// TIA Portal V19 export
DATA_BLOCK "A0302_Rulliera"   // DB85
// stored: InstanceOfName A0302_Rulliera_FB, InstanceOfType FB
"A0302_Rulliera_FB"
   // VAR_INPUT
   //    AreaInterface : "AreaInterface";
   //    ZSI : "udt_ZoneSafetyInterface";
   //    DSI_Feed1 : "udt_DeviceSafetyInterface";
   //    DSI_Feed2 : "udt_DeviceSafetyInterface";
   //    Drive_Ax1 : "TAx_DriveInterface";
   //    Drive_Ax2 : "TAx_DriveInterface";
   //    DataIn : Struct
   //       Ax : "SpeedMachine_DataIn";
   //       Sens : Struct
   //          Coda { ExternalAccessible := 'False'; ExternalVisible := 'False'; ExternalWritable := 'False'} : Struct
   //             FTC_Rall : Bool;
   //             FTC_Prox_Ing : Bool;
   //          END_STRUCT;
   //          Centro { ExternalAccessible := 'False'; ExternalVisible := 'False'; ExternalWritable := 'False'} : Struct
   //             FTC_Centrale : Bool;
   //          END_STRUCT;
   //       END_STRUCT;
   //    END_STRUCT;
   //    CIn { ExternalAccessible := 'False'; ExternalVisible := 'False'; ExternalWritable := 'False'} : Struct
   //       Manager : Struct
   //          Ax_1 : "SpeedMachine_CIn_Manager";
   //          Ax_2 : "SpeedMachine_CIn_Manager";
   //       END_STRUCT;
   //       SemiAut_Pb : Bool;
   //       P5 : Struct
   //          Sollevatori : "ValveMachine_COut";
   //          SpintoreLong : "ValveMachine_COut";
   //          Sens : Struct
   //             FTC_Ingombro_A0301 : Bool;
   //          END_STRUCT;
   //       END_STRUCT;
   //       Bordatrice : Struct
   //          StopBordatrice : Bool;
   //          ReadyForMove : Bool;
   //          StandbyBordatrice : Bool;
   //       END_STRUCT;
   //       Rulliera : Struct
   //          Centratori : "ValveMachine_COut";
   //          Sollevamento : "ValveMachine_COut";
   //          Coda : Struct
   //             Sens : Struct
   //                FTC_Rall : Bool;
   //                FTC_Prox_Ing : Bool;
   //             END_STRUCT;
   //          END_STRUCT;
   //          Centro : Struct
   //             Sens : Struct
   //                FTC_Centrale : Bool;
   //             END_STRUCT;
   //          END_STRUCT;
   //       END_STRUCT;
   //       CarroPareggCoda : Struct
   //          Ax : "Positioning_DOL_Machine_COut";
   //          Bloccaggio : "ValveMachine_COut";
   //          BattutaVerticale : "ValveMachine_COut";
   //          PareggiatoreLong : "ValveMachine_COut";
   //          Sens : Struct
   //             FTC_Ingombro_In : Bool;
   //             FTC_Ingombro_Out : Bool;
   //             PresenzaMat : Bool;
   //             PosPareggLong : Struct
   //                Value : LReal;
   //                CheckMeasure : Bool;
   //                Standstill : Bool;
   //             END_STRUCT;
   //          END_STRUCT;
   //       END_STRUCT;
   //       CarroPareggTesta : Struct
   //          Ax : "Positioning_DOL_Machine_COut";
   //          Bloccaggio : "ValveMachine_COut";
   //          Centraggio : "ValveMachine_COut";
   //          Sollevatore : "ValveMachine_COut";
   //          Sens : Struct
   //             FTC1_Rall : Bool;
   //             FTC2_Prox_Ls : Bool;
   //             PresenzaMat : Bool;
   //          END_STRUCT;
   //       END_STRUCT;
   //       BTrk : Struct
   //          ZoneA0302Entry_Empty : Bool;
   //          ZoneA0302Exit_Empty : Bool;
   //       END_STRUCT;
   //    END_STRUCT;
   //    Config : Struct
   //       Ax : "SpeedMachine_Config";
   //    END_STRUCT;
   //    HWID_Ax_TEL1 : Array[1..2] of HW_SUBMODULE;
   // END_VAR
   // VAR_OUTPUT
   //    MachineInterface : "MachineInterface";
   //    COut : Struct
   //       Ax_1 : "SpeedMachine_COut";
   //       Ax_2 : "SpeedMachine_COut";
   //       Ax_VelOveride : Struct
   //          Enable : Bool;
   //          Value : Real;
   //       END_STRUCT;
   //    END_STRUCT;
   // END_VAR
   // VAR_IN_OUT
   //    Par : Struct
   //       Ax : "SpeedMachine_Par";
   //       Ax_Aut : "A0301_Mach_Speed_Par";
   //    END_STRUCT;
   //    IEC_SP : Struct
   //       FTC_CodaRall : Struct
   //          TON_PT : Time;
   //          TOF_PT : Time;
   //       END_STRUCT;
   //       FTC_CodaProx_Ing : Struct
   //          TON_PT : Time;
   //          TOF_PT : Time;
   //       END_STRUCT;
   //       FTC_Centro : Struct
   //          TON_PT : Time;
   //          TOF_PT : Time;
   //       END_STRUCT;
   //    END_STRUCT;
   // END_VAR
   // VAR
   //    Alarm : Struct
   //       Rulliera : Array[1..2] of "SpeedMachine_Alr";
   //    END_STRUCT;
   //    Warning : Struct
   //       Rulliera : Array[1..2] of "SpeedMachine_Wng";
   //       OP_REST_MissingCnd : Bool;
   //       OP_WORK_MissingCnd : Bool;
   //    END_STRUCT;
   //    HMI : Struct
   //       Selection : Struct
   //          Ax : Int;
   //       END_STRUCT;
   //    END_STRUCT;
   //    Ax_1 : "SpeedMachine_FB";
   //    Ax_2 : "SpeedMachine_FB";
   //    ValueVelOvr { ExternalAccessible := 'False'; ExternalVisible := 'False'; ExternalWritable := 'False'} : Array[1..10] of Real;
   //    Sts : Struct
   //       OP_CanMoveFreely : Bool;
   //       OP_Bwd_Cnd : Bool;
   //       OP_Fwd_Cnd : Bool;
   //    END_STRUCT;
   //    Ctrl : Struct
   //       OP_Bwd_Man : Bool;
   //       OP_Fwd_Man : Bool;
   //       OP_Bwd_Aut : Bool;
   //       OP_Fwd_Aut : Bool;
   //       OP_Bwd_Run : Bool;
   //       OP_Fwd_Run : Bool;
   //    END_STRUCT;
   //    AUX : Struct
   //       OP_Bwd_PB : Bool;
   //       OP_Fwd_PB : Bool;
   //    END_STRUCT;
   //    TON_OP_REST_MissingCnd { S7_SetPoint := 'True'} : TON_TIME;
   //    TON_OP_WORK_MissingCnd { S7_SetPoint := 'True'} : TON_TIME;
   //    IEC_FTC_CodaRall : Struct
   //       TON_Delay : IEC_TIMER;
   //       TOF_Delay { S7_SetPoint := 'True'} : IEC_TIMER;
   //       FTC_On { S7_SetPoint := 'True'} : Bool;
   //    END_STRUCT;
   //    IEC_FTC_CodaProxIng : Struct
   //       TON_Delay : IEC_TIMER;
   //       TOF_Delay { S7_SetPoint := 'True'} : IEC_TIMER;
   //       FTC_On { S7_SetPoint := 'True'} : Bool;
   //    END_STRUCT;
   //    IEC_FTC_Centro : Struct
   //       TON_Delay : IEC_TIMER;
   //       TOF_Delay { S7_SetPoint := 'True'} : IEC_TIMER;
   //       FTC_On { S7_SetPoint := 'True'} : Bool;
   //    END_STRUCT;
   // END_VAR
BEGIN
END_DATA_BLOCK
